Yaskawa INFORM job: SYS_FILTER_CLEAN.JBI

/JOB
//NAME SYS_FILTER_CLEAN
//POS
///NPOS 0,0,0,0,0,0
//INST
///DATE 2022/11/09 10:44
///ATTR SC,RW
///GROUP1 RB1
NOP
DOUT OT#(2) ON
TIMER T=655.00
TIMER T=655.00
DOUT OT#(2) OFF
END
